FUNCTION_BLOCK FB_MotionAxisCommon IMPLEMENTS I_MotionAxisCommon
VAR_INPUT
END_VAR
VAR_OUTPUT
END_VAR
VAR
    {attribute 'no_copy'}
    AxisRef : REFERENCE TO AXIS_REF;
    // MC_ReadParameterSet Output
    {attribute 'hide'}
    mcReadParams: MC_ReadParameterSet;
    {attribute 'hide'}
    stAxisParameters: ST_AxisParameterSet;
    // NC Exposed Parameters
    {attribute 'hide'}
    stAxisParameterSetExposed : ST_AxisParameterSetExposed;
    {attribute 'hide'}
    bNcParamsReadInit   : BOOL;

    // NC er IO for ULINT (Biss-C)
    nRawEncoderULINT AT %I*: ULINT;
    // Raw encoder IO for UINT (Relative Encoders)
    nRawEncoderUINT AT %I*: UINT;
    // Raw encoder IO for INT (LVDT)
    nRawEncoderINT AT %I*: INT;
    // Raw encoder IO for INT (EL5072 LVDT)
    nRawEncoderDINT AT %I*: DINT;
    nEncoderCount	: UDINT;

    (* NC Blocks *)
    // MoveABsolute
    fbMcMoveAbsolute : MC_MoveAbsolute;
    bCommandedMoveAbsolute : BOOL;
    {attribute 'hide'}
    bMoveAbsoluteBusy : BOOL;
    {attribute 'hide'}
    bMoveAbsoluteDone : BOOL;
    {attribute 'hide'}
    bMoveAbsoluteError : BOOL;
    {attribute 'hide'}
    bCommandAborted : BOOL;
    {attribute 'hide'}
    nMoveAbsoluteErrorID : UDINT;
    // Reset
    fbMcReset 	: MC_Reset;
    {attribute 'hide'}
    bResetDone 	: BOOL;
    {attribute 'hide'}
    bResetBusy	: BOOL;
    {attribute 'hide'}
    bResetError	: BOOL;
    {attribute 'hide'}
    bResetErrorID	: UDINT;
    {attribute 'hide'}
    bReset		: BOOL;
    bCommandedReset : BOOL;

    // Power
    fbMcPower 		: MC_Power;
    bPowerEnable	: BOOL;
    bPowerEnablePositive : BOOL;
    bPowerEnableNegative : BOOL;
    {attribute 'hide'}
    bPowerIsEnabled : BOOL;
    {attribute 'hide'}
    bPowerBusy 		: BOOL;
    {attribute 'hide'}
    bPowerError 	: BOOL;
    {attribute 'hide'}
    nPowerErrorID 	: UDINT;
    {attribute 'hide'}
    fOverride 		: LREAL := 100.0;
    //////////////////
    fbMcHalt 		: MC_Halt;
    bCommandedHalt 	: BOOL;
    {attribute 'hide'}
    bHaltDone 		: BOOL;
    {attribute 'hide'}
    bHaltError 		: BOOL;
    {attribute 'hide'}
    nHaltErrorID 	: UDINT;
    {attribute 'hide'}
    bHaltBusy 		: BOOL;

    // Move parameters
    fMoveAbsoluteTargetPosition	: LREAL;
    fMoveAbsoluteTargetVelocity	: LREAL;
    fMoveAbsoluteTargetAcceleration	: LREAL := 0.0;
    fMoveAbsoluteTargetDeceleration	: LREAL := 0.0;
    fMoveAbsoluteTargetJerk	: LREAL := 0.0;
    nCommandLocal: UINT;
    nCmdDataLocal: UINT;
    eBufferMode	: MC_BufferMode := .MC_BufferMode.MC_Aborting;
    // Axis Status
    {attribute 'hide'}
    nAxisId : UDINT;
    {attribute 'hide'}
    fMeasuredVelocity : LREAL;
    {attribute 'hide'}
    fMeasuredPosition : LREAL;
    {attribute 'hide'}
    fMeasuredPositionDiff : LREAL;
    {attribute 'hide'}
    fMeasuredAcceleration : LREAL;
    // Needed for interlocks checks. please keep this as declared
    {attribute 'hide'}
    eAxisState : MC_AxisStates;
    // save and restore
    {attribute 'hide'}
    fbSetPos: MC_SetPosition;
    {attribute 'hide'}
    bClearPositionLag : BOOL := TRUE;
    {attribute 'hide'}
    bAxisError 		: BOOL;
    {attribute 'hide'}
    bPowerStatus 	: BOOL;
    {attribute 'hide'}
    bRestoreDone 	: BOOL;
    {attribute 'hide'}
    bRestoreError 	: BOOL;
    {attribute 'hide'}
    nRestoreErrorID : UDINT;

    // save and Restore
    {attribute 'hide'}
    RestoreTimer: TON;
    {attribute 'hide'}
    bRestoreInit: BOOL;
    {attribute 'hide'}
    bRestoreLoad: BOOL;
    {attribute 'hide'}
    nLatchError: UDINT;
    {attribute 'hide'}
    bEncError: BOOL;
    {attribute 'hide'}
    tRetryDelay: TIME := T#1S;
    {attribute 'hide'}
    nMaxRetries: UINT := 10;
    {attribute 'hide'}
    nCurrTries: UINT := 0;
    {attribute 'hide'}
    bRestoreWaitRetry: BOOL;
    {attribute 'hide'}
    tonRestoreRetry: TON;
    {attribute 'hide'}
    tRefreshTime : TIME := T#1S;

    // create a property for some of these
    {attribute 'hide'}
    bDone		: BOOL;
    {attribute 'hide'}
    bBusy		: BOOL;
    {attribute 'hide'}
    bInTargetPosition	: BOOL;

    // Error handling
    {attribute 'hide'}
    bError				: BOOL;
    {attribute 'hide'}
    nErrorId			: UDINT:=0;
    {attribute 'hide'}
    sErrorMessage		: STRING;
    {attribute 'hide'}
    ftDone 			: F_TRIG;
    {attribute 'hide'}
    ftStopExec 		: F_TRIG;
    {attribute 'hide'}
    rtTarget		: R_TRIG;
    {attribute 'hide'}
    rtHaltedDone	: R_TRIG;
    {attribute 'hide'}
    rtTargetReached	: R_TRIG;
    {attribute 'hide'}
    rtAbsoluteModeDone	: R_TRIG;

END_VAR

VAR PERSISTENT
    {attribute 'conditionalshow'}
    bSaved: BOOL;
    {attribute 'conditionalshow'}
    fSavedPosition: LREAL;
END_VAR

IF NOT __ISVALIDREF( AxisRef ) OR (THIS^.AxisRef.NcToPlc.AxisId = 0)THEN
    RETURN;
END_IF

////////////////////////////////////////////////////////////////////////
THIS^.AxisStatus();

THIS^.fbMcHalt(
    Axis := THIS^.AxisRef,
    Execute := THIS^.bCommandedHalt,
    Deceleration := fMoveAbsoluteTargetDeceleration,
    Jerk := fMoveAbsoluteTargetJerk,
    BufferMode := eBufferMode,
    Done => bHaltDone,
    Busy => bHaltBusy,
    CommandAborted => bCommandAborted,
    Error => bHaltError,
    ErrorID => nHaltErrorID
);

THIS^.bCommandedHalt := FALSE;

///////////////////////////////////////////////////////////////
// Reset the Axis based on signaling event on CommandedReset
//////////////////////////////////////////////////////////////
THIS^.fbMcReset(
    Axis := THIS^.AxisRef,
    Execute := THIS^.bCommandedReset,
    Done => bResetDone,
    Busy => bResetBusy,
    Error => bResetError,
    ErrorID => bResetErrorID,
);

IF bResetDone THEN
    THIS^.bCommandedReset := FALSE;
END_IF

//////////////////////////////////////////////////////////////////
// Power block depends on interlocks check in  iMotionInterlocks
/////////////////////////////////////////////////////////////////
THIS^.fbMcPower(
    Axis := THIS^.AxisRef,
    Enable := bPowerEnable,
    Enable_Positive := bPowerEnablePositive,
    Enable_Negative := bPowerEnableNegative,
    Override := fOverride,
    BufferMode := eBufferMode,
    (*Enabled*)
    Status => bPowerIsEnabled,
    Busy => bPowerBusy,
    Error => bPowerError,
    ErrorID => nPowerErrorID
);
////////////////////////////////////////////////////////////////////////////////////
// Handling Absolute move request using signaling events
// on CommandedMoveAbsolute
// clear the done bit after previous move is completed by an error condition
///////////////////////////////////////////////////////////////////////////////////
THIS^.fbMcMoveAbsolute(
    Axis := THIS^.AxisRef,
    Execute := THIS^.bCommandedMoveAbsolute,
    Position := fMoveAbsoluteTargetPosition,
    Velocity := fMoveAbsoluteTargetVelocity,
    Acceleration := fMoveAbsoluteTargetAcceleration,
    Deceleration := fMoveAbsoluteTargetDeceleration,
    Jerk := fMoveAbsoluteTargetJerk,
    BufferMode := eBufferMode,
    Done => ,
    Busy => bMoveAbsoluteBusy,
    Active => ,
    CommandAborted => bCommandAborted,
    Error => bMoveAbsoluteError,
    ErrorID => nMoveAbsoluteErrorID
);
////////////////////////////////////////////////////////////////////////////
// A neg edge on bMoveAbsoluteBusy comfirm that the previous move is done
//   either because of an error, an abort or a target reached.
//   bMoveAbsoluteDone will reset next cycle if done condition was an error
////////////////////////////////////////////////////////////////////////////
ftDone (CLK:=bMoveAbsoluteBusy);
IF ftDone.Q AND NOT bMoveAbsoluteError THEN
    bMoveAbsoluteDone := TRUE;

ELSIF AxisRef.Status.Error THEN
    bMoveAbsoluteDone := FALSE;
END_IF

THIS^.CalibrateRawEncValue();

THIS^.ErrorHandling();

THIS^.ExposeNCParams();
//////////////////////////////////////
// Handle save and restor
//////////////////////////////////////
THIS^.EncSaveRestore(bEnable:=TRUE);

{warning 'Add property implementation'}
PROPERTY AxisParameterSetExposed : ST_AxisParameterSetExposed
GET
AxisParameterSetExposed := stAxisParameterSetExposed;
END_GET
END_PROPERTY

{attribute 'monitoring':= 'variable'}
PROPERTY AxisState : MC_AxisStates
GET
AxisState := eAxisState;
END_GET
END_PROPERTY

METHOD AxisStatus
THIS^.AxisRef.ReadStatus();

(*Axis id in motion "motor"*)
nAxisId:=AxisRef.NcToPlc.AxisId;

(*Actual Velocity*)
fMeasuredVelocity:=AxisRef.NcToPlc.ActVelo;

(*Actual Position*)
IF AxisRef.Status.OpMode.Modulo THEN
    fMeasuredPosition:=AxisRef.NcToPlc.ModuloActPos;
ELSE
    fMeasuredPosition:=AxisRef.NcToPlc.ActPos;
END_IF

(*Actual Position Diff*)
fMeasuredPositionDiff:=AxisRef.NcToPlc.PosDiff;
(*Current Axis state*)
eAxisState := AxisRef.Status.MotionState;
(*Target Reached*)
bInTargetPosition := AxisRef.Status.InTargetPosition;
 (*Axis Error*)
bAxisError := AxisRef.Status.Error;
END_METHOD

PROPERTY BufferMode : MC_BufferMode
SET
eBufferMode := BufferMode;
END_SET
END_PROPERTY

{attribute 'monitoring':= 'variable'}
PROPERTY Busy : BOOL
GET
Busy := bBusy;
END_GET
END_PROPERTY

METHOD CalibrateRawEncValue
IF nRawEncoderULINT <> 0 THEN
    IF nRawEncoderULINT < 4294967296 THEN
        nEncoderCount := ULINT_TO_UDINT(nRawEncoderULINT);
    ELSE
        nEncoderCount := ULINT_TO_UDINT(18446744073709551615 - nRawEncoderULINT);
    END_IF
ELSIF nRawEncoderUINT <> 0 THEN
    nEncoderCount := UINT_TO_UDINT(nRawEncoderUINT);
ELSIF nRawEncoderINT <> 0 THEN
    nEncoderCount := INT_TO_UDINT(nRawEncoderINT);
ELSIF nRawEncoderDINT <> 0 THEN
    nEncoderCount := DINT_TO_UDINT(nRawEncoderDINT);
ELSE
    nEncoderCount := 0;
END_IF
END_METHOD

PROPERTY Cmd : UINT
SET
nCommandLocal := Cmd;
END_SET
END_PROPERTY

PROPERTY CmdData : UINT
SET
nCmdDataLocal := CmdData;
END_SET
END_PROPERTY

{attribute 'monitoring':= 'variable'}
PROPERTY CommandedHalt : BOOL
GET
 CommandedHalt := bCommandedHalt ;
END_GET
SET
 bCommandedHalt := CommandedHalt ;
END_SET
END_PROPERTY

{attribute 'monitoring':= 'variable'}
PROPERTY CommandedMoveAbsolute : BOOL
GET
 CommandedMoveAbsolute := bCommandedMoveAbsolute ;
END_GET
SET
 bCommandedMoveAbsolute := CommandedMoveAbsolute ;
END_SET
END_PROPERTY

{attribute 'monitoring':= 'variable'}
PROPERTY CommandedReset : BOOL
GET
CommandedReset := bCommandedReset;
END_GET
SET
CommandedReset := bCommandedReset;
END_SET
END_PROPERTY

METHOD EncErrorCheck : BOOL
VAR_INPUT
    EncError : BOOL;
    EncErrorCode : UDINT;
END_VAR
// Maybe different for some DS402 NC based drives. if so adjust or derive.
EncErrorCheck := EncError AND EncErrorCode >= 16#4400 AND EncErrorCode <= 16#44FF;
END_METHOD

{warning 'Add property implementation'}
PROPERTY EncoderCount : UDINT
GET
EncoderCount := nEncoderCount;
END_GET
END_PROPERTY

METHOD EncSaveRestore
VAR_INPUT
    bEnable : BOOL;
END_VAR
IF bEnable THEN
    // Trigger a load if anything was saved at all
    IF NOT bRestoreInit THEN
        bRestoreInit := TRUE;
        bRestoreLoad S= bSaved;
        fbSetPos.Options.ClearPositionLag := TRUE;
    END_IF

    // Set our position if bRestoreLoad is true
    fbSetPos( Axis:=THIS^.AxisRef, Execute:=bRestoreLoad, Position:=fSavedPosition);

    // Only load once, at startup
    bRestoreLoad R= fbSetPos.Done OR fbSetPos.Error;

    IF fbSetPos.Error THEN
        // Keep the error latched, it can disappear if Execute is set to FALSE
        nLatchError := fbSetPos.ErrorID;
        nCurrTries := nCurrTries + 1;
        IF nCurrTries >= nMaxRetries THEN
            // Alert the user that something has gone wrong
            bError := TRUE;
            nErrorId := nLatchError;
            sErrorMessage := 'Error loading previously saved position.';
        ELSE
            // Reset the FB for the next retry
            fbSetPos( Axis:=THIS^.AxisRef, Execute:=bRestoreLoad, Position:=fSavedPosition);
            // Try again
            bRestoreWaitRetry := TRUE;
        END_IF
    END_IF

    tonRestoreRetry( IN := bRestoreWaitRetry, PT := tRetryDelay);
    bRestoreLoad S= tonRestoreRetry.Q;
    bRestoreWaitRetry R= tonRestoreRetry.Q;

    // Check ST_MotionStage for an encoder error (range 0x44nn)
    bEncError:= AxisRef.Status.Error AND  ( AxisRef.Status.ErrorID  >= 16#4400  AND AxisRef.Status.ErrorID <= 16#44FF );
    // Do not save if we're currently loading or if there is an encoder error
    IF NOT bRestoreLoad AND NOT bEncError AND NOT bRestoreWaitRetry THEN
        fSavedPosition := fMeasuredPosition;
        // This persistent variable lets us check if anything was saved
        // It will be TRUE at startup if we have saved values
        bSaved := TRUE;
        (*
            use this with a timer of a change threshold on the fActPosition
            to trigger a save from this PLC program. otherwise this will be a spamming
            persistence, filling up the disk.
        *)
        // iPersistantDataStorage.TriggerWriteOfPersistentData := TRUE;
    END_IF
END_IF
END_METHOD

{attribute 'monitoring':= 'variable'}
PROPERTY Error : BOOL
GET
Error := bError;
END_GET
END_PROPERTY

METHOD ErrorHandling
(*Error from functions and Nc*)
IF fbMcPower.Error AND fbMcPower.Active THEN
    bError:=fbMcPower.Enable;
    nErrorId:=fbMcPower.ErrorID;
ELSIF AxisRef.Status.Error  THEN
    bError:=TRUE;
    nErrorId:=AxisRef.Status.ErrorID;
ELSIF fbMcMoveAbsolute.Error (*fbMcMoveAbsolute.Active*) THEN
    bError:=fbMcMoveAbsolute.Execute;
    nErrorId:=fbMcMoveAbsolute.ErrorID;
ELSIF fbMcHalt.Error AND fbMcHalt.Active THEN
    bError:=fbMcHalt.Execute;
    nErrorId:=fbMcHalt.ErrorID;
ELSIF fbMcReset.Error  THEN
    bError:=fbMcPower.Enable;
    nErrorId:=fbMcPower.ErrorID;
ELSE
    bError:=FALSE;
    nErrorId:=0;
END_IF;
END_METHOD

{attribute 'monitoring':= 'variable'}
PROPERTY ErrorID : UDINT
GET
ErrorID := nErrorId;
END_GET
END_PROPERTY

{attribute 'monitoring':= 'variable'}
PROPERTY ErrorMessage : STRING
GET
ErrorMessage := sErrorMessage;
END_GET
END_PROPERTY

METHOD ExposeNCParams : BOOL;

VAR_INST
    timer: TON;
    bExecute: BOOL := TRUE;
    nLatchErrId: UDINT;
END_VAR
timer( IN:= NOT bExecute, PT:=tRefreshTime);

bExecute S= timer.Q;
mcReadParams(
    Parameter:=THIS^.stAxisParameters,
    Axis:= AxisRef,
    Execute:= bExecute );

IF mcReadParams.Error THEN
    bError := TRUE;
    nErrorID := mcReadParams.ErrorID;
    // Log this error
END_IF

(* IF mcReadParams.ErrorID <> 0 THEN
    nLatchErrId := 0;
END_IF *)

// Copy axis parameters that we want to expose to the EPICS layer.
THIS^.stAxisParameterSetExposed.bCtrlEnablePosDiffControl     := THIS^.stAxisParameters.bCtrlEnablePosDiffControl;
THIS^.stAxisParameterSetExposed.bEncEnableSoftEndMaxControl   := THIS^.stAxisParameters.bEncEnableSoftEndMaxControl;
THIS^.stAxisParameterSetExposed.bEncEnableSoftEndMinControl   := THIS^.stAxisParameters.bEncEnableSoftEndMinControl;
THIS^.stAxisParameterSetExposed.fAccelerationMax              := THIS^.stAxisParameters.fAccelerationMax;
THIS^.stAxisParameterSetExposed.fCtrlPosDiffMax               := THIS^.stAxisParameters.fCtrlPosDiffMax;
THIS^.stAxisParameterSetExposed.fCtrlPosDiffMaxTime           := THIS^.stAxisParameters.fCtrlPosDiffMaxTime;
THIS^.stAxisParameterSetExposed.fDecelerationMax              := THIS^.stAxisParameters.fDecelerationMax;
THIS^.stAxisParameterSetExposed.fEncSoftEndMax                := THIS^.stAxisParameters.fEncSoftEndMax;
THIS^.stAxisParameterSetExposed.fEncSoftEndMin                := THIS^.stAxisParameters.fEncSoftEndMin;
THIS^.stAxisParameterSetExposed.fVeloMaximum                  := THIS^.stAxisParameters.fVeloMaximum;
THIS^.stAxisParameterSetExposed.fEncOffset               	  := THIS^.stAxisParameters.fEncOffset;
THIS^.stAxisParameterSetExposed.fEncScaleFactorInternal       := THIS^.stAxisParameters.fEncScaleFactorInternal;

bExecute R= mcReadParams.Done OR mcReadParams.Error;
bNCParamsReadInit S= mcReadParams.Done;
END_METHOD

//FB_Init is always available implicitly and it is used primarily for initialization.
//The return value is not evaluated. For a specific influence, you can also declare the
//methods explicitly and provide additional code there with the standard initialization
//code. You can evaluate the return value.
METHOD FB_Init: BOOL
VAR_INPUT
    bInitRetains: BOOL; // TRUE: the retain variables are initialized (reset warm / reset cold)
    bInCopyCode: BOOL;  // TRUE: the instance will be copied to the copy code afterward (online change)
    AxisReference : REFERENCE TO AXIS_REF;
END_VAR
THIS^.AxisRef REF= AxisReference;
END_METHOD

PROPERTY HaltBusy : BOOL
GET
HaltBusy := bHaltBusy;
END_GET
END_PROPERTY

PROPERTY HaltDone : BOOL
GET
HaltDone := bHaltDone;
END_GET
END_PROPERTY

{warning 'Add property implementation'}
PROPERTY HaltError : BOOL
GET
HaltError := bHaltError;
END_GET
END_PROPERTY

PROPERTY HaltErrorID : UDINT
GET
HaltErrorID := nHaltErrorID;
END_GET
END_PROPERTY

{attribute 'monitoring':= 'variable'}
PROPERTY InTargetPosition : BOOL
GET
InTargetPosition := bInTargetPosition;
END_GET
END_PROPERTY

{warning 'Add method implementation '}
METHOD InterruptMove
END_METHOD

{attribute 'monitoring':= 'variable'}
PROPERTY MeasuredAcceleration : LREAL
GET
MeasuredAcceleration := fMeasuredAcceleration;
END_GET
END_PROPERTY

{attribute 'monitoring':= 'variable'}
PROPERTY MeasuredPosition : LREAL
GET
MeasuredPosition := fMeasuredPosition;
END_GET
END_PROPERTY

{attribute 'monitoring':= 'variable'}
PROPERTY MeasuredPositionDiff : LREAL
GET
MeasuredPositionDiff := fMeasuredPositionDiff;
END_GET
END_PROPERTY

{attribute 'monitoring':= 'variable'}
PROPERTY MeasuredVelocity : LREAL
GET
 MeasuredVelocity := MeasuredVelocity;
END_GET
END_PROPERTY

{warning 'Add property implementation'}
PROPERTY ModeOfOperation : SINT
GET
END_GET
SET
END_SET
END_PROPERTY

{warning 'Add property implementation'}
PROPERTY MoveAbsoluteBusy : BOOL
GET
MoveAbsoluteBusy := bMoveAbsoluteBusy;
END_GET
END_PROPERTY

PROPERTY MoveAbsoluteDone : BOOL
GET
MoveAbsoluteDone := bMoveAbsoluteDone;
END_GET
END_PROPERTY

PROPERTY MoveAbsoluteError : BOOL
GET
MoveAbsoluteError := bMoveAbsoluteError;
END_GET
END_PROPERTY

PROPERTY MoveAbsoluteErrorID : UDINT
GET
MoveAbsoluteErrorID := nMoveAbsoluteErrorID ;
END_GET
END_PROPERTY

{attribute 'monitoring':= 'variable'}
PROPERTY MoveAbsoluteTargetAcceleration : LREAL
GET
MoveAbsoluteTargetAcceleration := fMoveAbsoluteTargetAcceleration;
END_GET
SET
fMoveAbsoluteTargetAcceleration := MoveAbsoluteTargetAcceleration;
END_SET
END_PROPERTY

{attribute 'monitoring':= 'variable'}
PROPERTY MoveAbsoluteTargetDeceleration : LREAL
GET
MoveAbsoluteTargetDeceleration := fMoveAbsoluteTargetDeceleration;
END_GET
SET
END_SET
END_PROPERTY

{attribute 'monitoring':= 'variable'}
PROPERTY MoveAbsoluteTargetJerk : LREAL
GET
MoveAbsoluteTargetJerk := fMoveAbsoluteTargetJerk;
END_GET
SET
fMoveAbsoluteTargetJerk := MoveAbsoluteTargetJerk;
END_SET
END_PROPERTY

{attribute 'monitoring':= 'variable'}
PROPERTY MoveAbsoluteTargetPosition : LREAL
GET
fMoveAbsoluteTargetPosition := MoveAbsoluteTargetPosition ;
END_GET
SET
MoveAbsoluteTargetPosition  := fMoveAbsoluteTargetPosition;
END_SET
END_PROPERTY

{attribute 'monitoring':= 'variable'}
PROPERTY MoveAbsoluteTargetVelocity : LREAL
GET
MoveAbsoluteTargetVelocity := fMoveAbsoluteTargetVelocity;
END_GET
SET
fMoveAbsoluteTargetVelocity := MoveAbsoluteTargetVelocity;
END_SET
END_PROPERTY

PROPERTY NCParamsReadInit : BOOL
GET
NCParamsReadInit := bNCParamsReadInit;
END_GET
END_PROPERTY

{warning 'Add property implementation'}
PROPERTY NegativeMotionIsEnabled : BOOL
GET
END_GET
END_PROPERTY

{warning 'Add property implementation'}
PROPERTY PositiveMotionIsEnabled : BOOL
GET
END_GET
END_PROPERTY

PROPERTY PowerEnable : BOOL
GET
PowerEnable := bPowerEnable;
END_GET
SET
bPowerEnable := PowerEnable;
END_SET
END_PROPERTY

PROPERTY PowerEnableNegative : BOOL
GET
PowerEnableNegative := bPowerEnableNegative;
END_GET
SET
bPowerEnableNegative := PowerEnableNegative;
END_SET
END_PROPERTY

PROPERTY PowerEnablePositive : BOOL
GET
PowerEnablePositive := bPowerEnablePositive;
END_GET
SET
bPowerEnablePositive := PowerEnablePositive;
END_SET
END_PROPERTY

PROPERTY PowerError : BOOL
GET
PowerError := bPowerError;
END_GET
END_PROPERTY

PROPERTY PowerErrorID : UDINT
GET
PowerErrorID  := nPowerErrorID;
END_GET
END_PROPERTY

{attribute 'monitoring':= 'variable'}
PROPERTY PowerIsEnabled : BOOL
GET
PowerIsEnabled := bPowerIsEnabled;
END_GET
END_PROPERTY

{warning 'Add property implementation'}
PROPERTY PowerOverride : LREAL
GET
PowerOverride := fOverride;
END_GET
SET
fOverride := PowerOverride;
END_SET
END_PROPERTY

PROPERTY PowerStatus : BOOL
GET
PowerStatus := bPowerStatus;
END_GET
END_PROPERTY

{warning 'Add property implementation'}
PROPERTY RefreshDelay : TIME
GET
RefreshDelay := tRefreshTime;
END_GET
SET
tRefreshTime := RefreshDelay;
END_SET
END_PROPERTY

{warning 'Add method implementation '}
METHOD Reset
END_METHOD

PROPERTY ResetBusy : BOOL
GET
ResetBusy := bResetBusy;
END_GET
END_PROPERTY

PROPERTY ResetDone : BOOL
GET
ResetDone := bResetDone;
END_GET
END_PROPERTY

PROPERTY ResetError : BOOL
GET
ResetError := bResetError ;
END_GET
END_PROPERTY

PROPERTY ResetErrorID : UDINT
GET
ResetErrorID := bResetErrorID ;
END_GET
END_PROPERTY

{attribute 'monitoring':= 'variable'}
PROPERTY RestoreDone : BOOL
GET
RestoreDone := bRestoreDone;
END_GET
END_PROPERTY

{attribute 'monitoring':= 'variable'}
PROPERTY RestoreError : BOOL
GET
RestoreError := bRestoreError;
END_GET
END_PROPERTY

{attribute 'monitoring':= 'variable'}
PROPERTY RestoreErrorID : UDINT
GET
RestoreErrorID := nRestoreErrorID;
END_GET
END_PROPERTY

{warning 'Add property implementation'}
PROPERTY Servo : BOOL
GET
END_GET
SET
END_SET
END_PROPERTY

{warning 'Add method implementation '}
(*
    Check all post condition before updating bCommandedMoveAbsolute
    The implmentatation will depend on the axis type
    DS402 NC/Direct axis : Implementation need to check that the drive is in the correct mode before initaiting the move then set bCommandedMoveAbsolute
    MP NC axis : will immediately write to bCommandedMoveAbsolute
*)
METHOD StartMove
END_METHOD

{warning 'Add method implementation '}
METHOD StopMove
END_METHOD

END_FUNCTION_BLOCK

(* stored: Version 1.1.0.1
   POU FB_MotionAxisCommon: Id {b2f4c148-bcde-4ca5-a7a9-abd4413ce8ab}, SpecialFunc None
   Property AxisParameterSetExposed: Id {bd38f88c-c219-4363-856f-6d4d63c13ec4}
   Get Get: Id {50330633-1a97-458e-b8ef-ffa028d8a61b}
   Property AxisState: Id {74147cdb-4b8a-4b74-a37f-eaadafea6e7a}
   Get Get: Id {5079f451-585f-45fc-ac12-d15b6be4da3e}
   Method AxisStatus: Id {a2f51608-f018-4206-8683-35f8a139b286}
   Property BufferMode: Id {bbbbad1c-a25b-4e16-b8e7-df89fde7223f}
   Set Set: Id {09436c45-d463-45eb-84c8-25add90ecfb1}
   Property Busy: Id {dbe7370a-96f9-4293-8d7a-aa83479a93ec}
   Get Get: Id {cf057b51-ea7a-4a6d-80b9-c1ff9ed546dd}
   Method CalibrateRawEncValue: Id {1731f1b4-fc8d-48cd-81d7-d75b2a571773}
   Property Cmd: Id {30a03909-94ab-4c48-bbf6-b0a60851a6e1}
   Set Set: Id {6c0d67c1-1597-4c36-b826-df5509e470ed}
   Property CmdData: Id {7ff40bd6-da45-4dd0-ab0a-405875312520}
   Set Set: Id {8b8d023c-647c-4ba1-9343-2904408a7d08}
   Property CommandedHalt: Id {5701fdc8-2e51-4874-9fa9-19bda9807780}
   Get Get: Id {58543ccd-d922-4229-9442-293feb0d6152}
   Set Set: Id {7ed3e647-a081-4cb2-8f34-db13ffc4a31b}
   Property CommandedMoveAbsolute: Id {c5f400b9-3987-40e0-abc8-1ea7986ea753}
   Get Get: Id {6225139f-92d7-4d2a-a472-e9a3b670bd69}
   Set Set: Id {02f2da0e-7628-484b-9d3e-26ee273505a0}
   Property CommandedReset: Id {d14f3271-8a4e-47d2-a6e5-bf876ab86a15}
   Get Get: Id {4d839e9d-2767-406e-adbb-ee037ab384eb}
   Set Set: Id {83e91627-4943-4145-bd4f-770ab6240427}
   Method EncErrorCheck: Id {7c7bd705-a252-45ea-8394-e497101ce9be}
   Property EncoderCount: Id {5225d004-dac1-4dfa-90f6-2aa283ea59c1}
   Get Get: Id {4699599a-607a-4379-8415-7f67e45880a3}
   Method EncSaveRestore: Id {f9f7cdfc-d8df-423b-8c50-6f118d29a052}
   Property Error: Id {2819c2f0-b6fd-42b1-b42d-175038209c48}
   Get Get: Id {c757a456-f781-4926-9229-39a5572ee16c}
   Method ErrorHandling: Id {e3e9f4c3-bd6f-4479-80bb-9cc735eca053}
   Property ErrorID: Id {b7569608-1ea8-4914-a3b4-543b15f7c860}
   Get Get: Id {37935438-07d0-4e35-a5a0-50e5e1f3d03b}
   Property ErrorMessage: Id {66fe07db-5064-463d-8bc4-a9cd6438f037}
   Get Get: Id {9aa0784b-8730-40a7-875e-aca2a5851c4c}
   Method ExposeNCParams: Id {dd5f801a-4004-4e64-a8a8-d3052d398ddb}
   Method FB_Init: Id {8bc50fb9-2f4e-4094-860c-18b3654dc16c}
   Property HaltBusy: Id {3729316f-44b8-4fc4-a4b3-679c26ec4375}
   Get Get: Id {73cbbd46-fd66-47f4-add3-798f531a9bfa}
   Property HaltDone: Id {aad1e7f5-ccd7-40f9-ad49-dcb715adbd3c}
   Get Get: Id {4f30d372-5e5c-43d7-85b0-a3893ab82baf}
   Property HaltError: Id {122f2f3a-178e-4ab7-b626-63e0bfb3c34a}
   Get Get: Id {26b0f530-f1ab-41f4-9a14-5442f2137687}
   Property HaltErrorID: Id {3b38681c-deb8-4f04-81e3-6de42841d4b4}
   Get Get: Id {2fe75d12-42ba-4a63-baee-0a8ed41cccbe}
   Property InTargetPosition: Id {8b3da1a3-aac2-42ca-9975-d233f7ffa27f}
   Get Get: Id {f0a1ade3-7297-4a8f-beb4-690092869c39}
   Method InterruptMove: Id {984711c6-7ff8-4f68-a02c-bc123018017f}
   Property MeasuredAcceleration: Id {851053ea-382f-4583-9e4d-2b1276874669}
   Get Get: Id {a1b55aca-d249-4132-a71f-1a170a4acdb1}
   Property MeasuredPosition: Id {a1cdbee3-0442-4424-9073-d6b393fb281e}
   Get Get: Id {62651479-095e-41cf-8939-2596a39a209d}
   Property MeasuredPositionDiff: Id {6f86c803-2111-484d-b5ed-4bedcd28495d}
   Get Get: Id {739aeb9c-249b-4194-bbb7-977990ba22fa}
   Property MeasuredVelocity: Id {7b6c331a-cfef-459b-88c0-ee39dd85009c}
   Get Get: Id {59076a82-9603-464d-9a99-a7944ba41d31}
   Property ModeOfOperation: Id {8eb0be67-7b04-4f8a-9914-0cbc01ce3595}
   Get Get: Id {a63d16eb-be98-4f86-8cb3-59daccc0bae8}
   Set Set: Id {41247b41-02ec-4aa7-9799-8371c49df1dc}
   Property MoveAbsoluteBusy: Id {8bba339d-272b-4575-bd5a-b3466a6e1c1c}
   Get Get: Id {cdf62e84-f8c6-4d30-bda2-e0acfc8d7692}
   Property MoveAbsoluteDone: Id {f9843104-9697-4366-9d0a-efa68a9fe9cf}
   Get Get: Id {8c9450f2-f665-4820-8191-e495b60638d7}
   Property MoveAbsoluteError: Id {743da600-6237-4d55-ac5c-8914ead4576f}
   Get Get: Id {e265747d-1e09-43c3-a937-bb427300328a}
   Property MoveAbsoluteErrorID: Id {81230976-e371-4bd9-9ed8-1beab6098570}
   Get Get: Id {5b0490c3-6dda-431e-981a-1cc69dcf77c7}
   Property MoveAbsoluteTargetAcceleration: Id {23311078-e7b9-4732-95b1-14c4c940a48c}
   Get Get: Id {30e1e061-024a-4d41-b2b4-6cdae17efcf8}
   Set Set: Id {c5e020e7-b0f8-4ce9-8272-4643af10c97a}
   Property MoveAbsoluteTargetDeceleration: Id {ea6189c7-6f42-4b41-b1c5-136e6340b80d}
   Get Get: Id {62f6fac2-c751-4c95-9e3f-c5a1b02e7a66}
   Set Set: Id {9e90be87-2eaa-49e4-9cfe-63e58373720a}
   Property MoveAbsoluteTargetJerk: Id {feefd4b1-94bf-447b-ab77-5646e681427f}
   Get Get: Id {f61c8aa4-6897-44f1-ae86-bde4382d02e3}
   Set Set: Id {637957fd-52a7-47f8-be67-da716da31c5c}
   Property MoveAbsoluteTargetPosition: Id {a6a2bcd1-7250-4b42-a6c3-9ba60983fbf1}
   Get Get: Id {74ecfcba-8315-4658-96b3-13327f7fbb7f}
   Set Set: Id {6c1082d7-96f3-4f8a-907d-c5d126db8bcc}
   Property MoveAbsoluteTargetVelocity: Id {9fd3f074-657b-4292-9885-57bed5f0b5b5}
   Get Get: Id {4ad245ec-4d06-4905-9c1d-24c221eef44e}
   Set Set: Id {87319ed5-2102-4b4f-9d55-bc59fbcc2970}
   Property NCParamsReadInit: Id {fc8144c2-ca29-4700-853c-a4a1e0fc319a}
   Get Get: Id {bf6c53f4-cc0b-4a81-96a0-d612250516fd}
   Property NegativeMotionIsEnabled: Id {b056ba37-46d4-430c-b297-3429bcd88dfb}
   Get Get: Id {38017209-5853-4f40-9d9e-0296332f7117}
   Property PositiveMotionIsEnabled: Id {ea12efb9-bcaa-4d5b-b6e2-2e2dc3b6153d}
   Get Get: Id {e5de1c9d-829b-4c5b-ae62-c664d60724eb}
   Property PowerEnable: Id {52a6864f-72c8-4689-b02e-2c6a93a6e57f}
   Get Get: Id {48500b16-0ce2-49f1-b21f-0533cc814246}
   Set Set: Id {0e7b72f0-3056-4080-bb7d-d6320654a326}
   Property PowerEnableNegative: Id {9f868447-67ce-4fa8-8603-0d81dd8e16f8}
   Get Get: Id {f8c49fa2-7312-4ebe-af66-a98a5b908ac7}
   Set Set: Id {f24d0b9a-f4f2-4458-a840-c6a1e2d1997b}
   Property PowerEnablePositive: Id {506de153-294e-4bda-a0dc-d37860a787f4}
   Get Get: Id {17b9d9b0-adc5-40b4-bdc8-ed9f3db477a3}
   Set Set: Id {0289db3a-85be-4799-a43b-dfa6f8e142a2}
   Property PowerError: Id {539da31b-05fd-42ae-90e9-cbefc3f2bcac}
   Get Get: Id {b7dcf07b-fc82-41ed-8ef8-6b0d511db94d}
   Property PowerErrorID: Id {0bd4689a-ceb9-4b34-96ab-62db6e708dc9}
   Get Get: Id {8c377cae-9b9a-4798-9990-ce542ac2a885}
   Property PowerIsEnabled: Id {c941a8e7-00f0-444d-978a-92a197132d8b}
   Get Get: Id {2d6397d6-01f1-41c2-a5ef-435d083bd604}
   Property PowerOverride: Id {b3b04403-4328-4a31-87db-cdf6d088144b}
   Get Get: Id {2fcfe7b8-ee2d-413f-adb0-61ee2d9519f2}
   Set Set: Id {23e4495f-08f9-44cc-875e-75e265ee63c5}
   Property PowerStatus: Id {8c236779-ba9c-4491-b5ea-5964867bf7ba}
   Get Get: Id {68f8524d-3388-4d1d-af05-c26bf9bb6cb3}
   Property RefreshDelay: Id {c668952b-b953-4bf4-ba2d-d28533b1ae8e}
   Get Get: Id {6c1f6886-4ab3-4ece-8855-4a22fb749cdc}
   Set Set: Id {9eb9790d-2215-40d1-8644-3da2d9a87714}
   Method Reset: Id {6a2ae321-d961-46f9-9ef7-70fbe99ba833}
   Property ResetBusy: Id {8142dd1d-e6ed-48f9-82bc-40d844e67918}
   Get Get: Id {ae505aa3-2b34-4b62-baf6-2dd558f81f4c}
   Property ResetDone: Id {3d5f9615-daf8-4aa9-9a70-1301f4ad44e0}
   Get Get: Id {83ba80a6-41e7-4816-a119-f9c2b92e0fc3}
   Property ResetError: Id {f9435560-a022-4839-9f1b-c67ce2725041}
   Get Get: Id {611a12af-6d97-4231-8e80-6dfa5c281869}
   Property ResetErrorID: Id {6eae6dee-1d7f-4456-bada-6c7d64b47385}
   Get Get: Id {2046024e-9bc7-48c7-b98e-aff6b96909a8}
   Property RestoreDone: Id {1c7ebab8-bf9d-41be-8ae1-4fa486ea2515}
   Get Get: Id {8bb5e119-978e-4082-b448-c991ff07ea58}
   Property RestoreError: Id {c8bc283c-88b2-4008-a719-c60968bbb480}
   Get Get: Id {1b3bfbf0-a349-43d3-aecc-31567f65bb93}
   Property RestoreErrorID: Id {c4c8ceda-d787-48c0-a1bc-b70a886d9e03}
   Get Get: Id {f56d3cf0-c7fc-49f9-b8b1-9feae45afdc2}
   Property Servo: Id {82295e5d-c599-4c17-9ce3-d6526bb012d0}
   Get Get: Id {af265e1e-e217-4bdc-8c1f-114ac95a5662}
   Set Set: Id {1762397d-0720-43cf-b640-81833e5fa3ab}
   Method StartMove: Id {7a80712e-d5dd-4474-a636-e52dbc5f0821}
   Method StopMove: Id {3b6ba44c-ffc1-4359-9996-2aa25ffb1a6f} *)
